FUNCTION Convert_TOD_TO_WORD : Hresult
VAR_INPUT
	in : TOD;
	out : REFERENCE TO WORD;
END_VAR
VAR
	converted : WORD;
END_VAR
VAR CONSTANT
	INCOMPATIBLE : HRESULT := 16#9811070E;
END_VAR

converted := TOD_TO_WORD(in);

IF (WORD_TO_TOD(converted) <> in) THEN
	Convert_TOD_TO_WORD := INCOMPATIBLE;
	RETURN;
END_IF

out := converted;

END_FUNCTION

(* stored: Version 1.1.0.1, ProductVersion 3.1.4024.12
   POU Convert_TOD_TO_WORD: Id {8407c5e1-4d35-4fb9-b4a6-2b1140298dee}, SpecialFunc None *)
